PROGRAM ProgramSequence
VAR
	X: INT;
END_VAR

IF NOT GVL.System_Start_Stop THEN
	X := 10;
	GVL.Motor1_State := 0;
	GVL.Motor2_State := 0;	
END_IF

	CASE X OF
0: IF NOT GVL.Motor1_State THEN
 	GVL.Motor1_State := 1;
	X := 1;
	END_IF
	
1: IF GVL.SensorInput = 1 THEN
	GVL.Motor2_Direction := 0;
	GVL.Motor2_State := 1;
	GVL.ProductA_Amount := GVL.ProductA_Amount + 1;
	X := 2;
	ELSIF GVL.SensorInput = 2 THEN
	GVL.Motor2_Direction := 1;
	GVL.Motor2_State := 1;
	X := 2;
	GVL.ProductB_Amount := GVL.ProductB_Amount + 1;
	END_IF
	
2: 	GVL.Motor1_State := 0;
	IF GVL.Conveyor2_Free THEN
	X := 0;
	END_IF
	END_CASE

END_PROGRAM

(* stored: Version 1.1.0.1, ProductVersion 3.1.4024.12
   POU ProgramSequence: Id {57073d3a-1ff5-4cda-8931-755335b396bf}, SpecialFunc None *)
